FUNCTION_BLOCK WorkPieces (* Composite Function Block Type *)
  (* Standard: 61499-2 *)
  (* Version 0.0, 7/14/2016, Andrei, nxtControl GmbH, template *)
  PACKAGE Main;
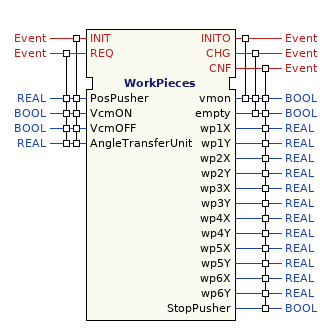
  EVENT_INPUT
    INIT WITH PosPusher, AngleTransferUnit, VcmON, VcmOFF; (* Initialization Request *)
    REQ WITH PosPusher, AngleTransferUnit, VcmON, VcmOFF; (* Normal Execution Request *)
  END_EVENT
  EVENT_OUTPUT
    INITO WITH vmon; (* Initialization Confirm *)
    CHG WITH vmon, empty;
    CNF WITH vmon, empty, wp1X, wp1Y, wp2X, wp2Y, wp3X, wp3Y, wp4X, wp4Y, wp5X, wp5Y, wp6X, wp6Y, StopPusher; (* Execution Confirmation *)
  END_EVENT
  VAR_INPUT
    PosPusher : REAL; (* Input event qualifier *)
    VcmON : BOOL;
    VcmOFF : BOOL;
    AngleTransferUnit : REAL;
  END_VAR
  VAR_OUTPUT
    vmon : BOOL; (* Output event qualifier *)
    empty : BOOL;
    wp1X : REAL;
    wp1Y : REAL;
    wp2X : REAL;
    wp2Y : REAL;
    wp3X : REAL;
    wp3Y : REAL;
    wp4X : REAL;
    wp4Y : REAL;
    wp5X : REAL;
    wp5Y : REAL;
    wp6X : REAL;
    wp6Y : REAL;
    StopPusher : BOOL;
  END_VAR
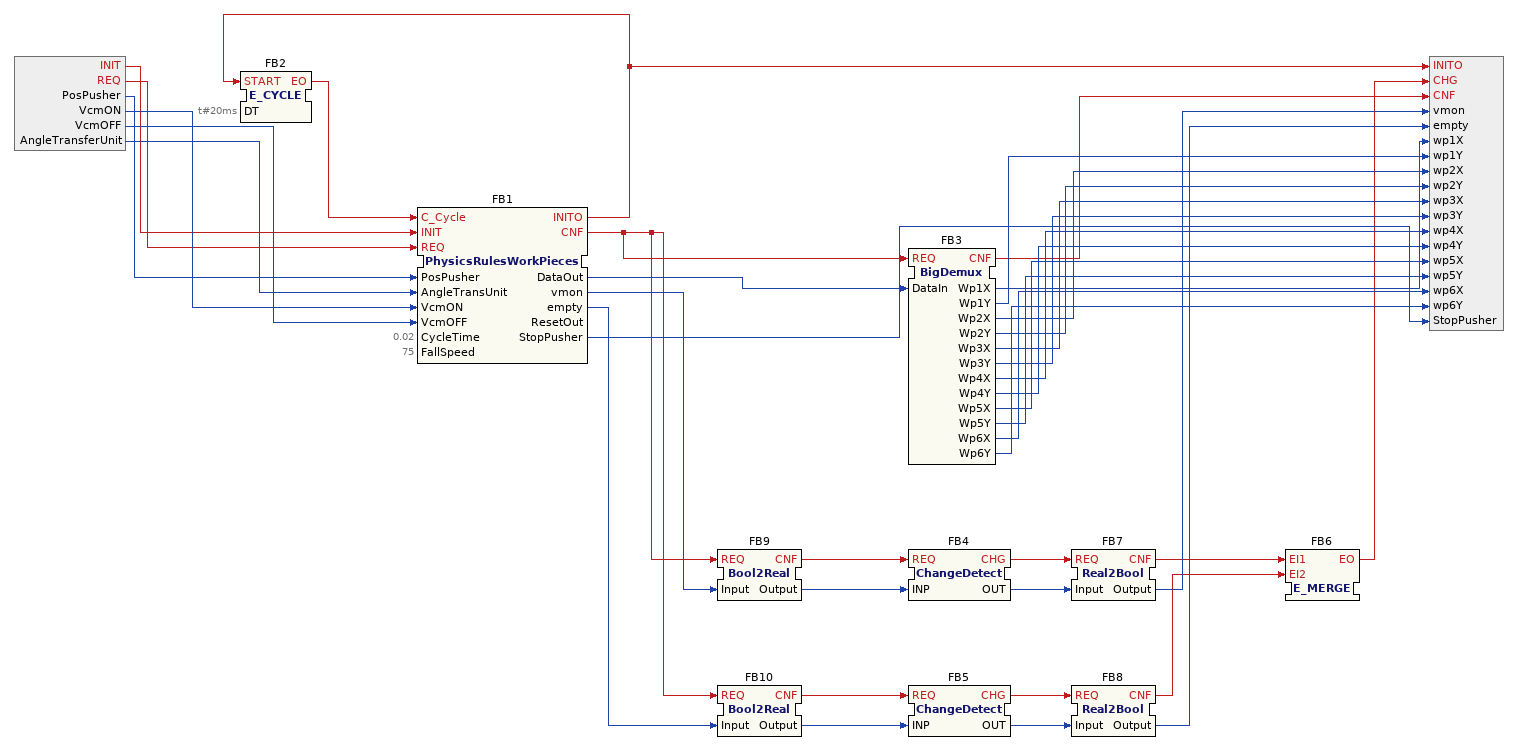
  FBS
    FB2 : E_CYCLE(DT := t#20ms);
    FB4 : ChangeDetect;
    FB5 : ChangeDetect;
    FB6 : E_MERGE;
    FB3 : BigDemux;
    FB1 : PhysicsRulesWorkPieces(CycleTime := 0.02, FallSpeed := 75);
    FB7 : Real2Bool;
    FB8 : Real2Bool;
    FB9 : Bool2Real;
    FB10 : Bool2Real;
  END_FBS
  EVENT_CONNECTIONS
    INIT TO FB1.INIT;
    REQ TO FB1.REQ;
    FB2.EO TO FB1.C_Cycle;
    FB1.CNF TO FB3.REQ;
    FB4.CHG TO FB7.REQ;
    FB5.CHG TO FB8.REQ;
    FB6.EO TO CHG;
    FB1.CNF TO FB9.REQ;
    FB1.CNF TO FB10.REQ;
    FB3.CNF TO CNF;
    FB1.INITO TO INITO;
    FB1.INITO TO FB2.START;
    FB7.CNF TO FB6.EI1;
    FB8.CNF TO FB6.EI2;
    FB9.CNF TO FB4.REQ;
    FB10.CNF TO FB5.REQ;
  END_CONNECTIONS
  DATA_CONNECTIONS
    PosPusher TO FB1.PosPusher;
    AngleTransferUnit TO FB1.AngleTransUnit;
    VcmON TO FB1.VcmON;
    VcmOFF TO FB1.VcmOFF;
    FB1.DataOut TO FB3.DataIn;
    FB4.OUT TO FB7.Input;
    FB5.OUT TO FB8.Input;
    FB1.vmon TO FB9.Input;
    FB1.empty TO FB10.Input;
    FB3.Wp1X TO wp1X;
    FB3.Wp1Y TO wp1Y;
    FB3.Wp2X TO wp2X;
    FB3.Wp2Y TO wp2Y;
    FB3.Wp3X TO wp3X;
    FB3.Wp3Y TO wp3Y;
    FB3.Wp4X TO wp4X;
    FB3.Wp4Y TO wp4Y;
    FB3.Wp5X TO wp5X;
    FB3.Wp5Y TO wp5Y;
    FB3.Wp6X TO wp6X;
    FB3.Wp6Y TO wp6Y;
    FB1.StopPusher TO StopPusher;
    FB7.Output TO vmon;
    FB8.Output TO empty;
    FB9.Output TO FB4.INP;
    FB10.Output TO FB5.INP;
  END_CONNECTIONS
END_FUNCTION_BLOCK
